Universal Robots URScript: dus_init.script

# =============================================================================
#  dus_init.script — dusan_v1
#  파라미터를 읽고 피치·행수를 계산한다. 실시간 발행 스레드를 띄운다
#
#  펜던트에서 "1_init" 자리에 스크립트 노드를 파일(File) 모드로 넣고 지정한다.
#
#  ※ def main() 으로 감싸지 말 것 (펜던트가 호출하지 않는다)
#  ※ 최상위에 global 을 쓰지 말 것 (preamble 이 이미 선언·대입해 뒀다)
#  ※ if / while 은 반드시 end 로 닫을 것
# =============================================================================

def ini_w1(a, v):
    if (v > 32000):
        v = 32000
    end
    if (v < -32000):
        v = -32000
    end
    write_port_register(a, floor(v + 0.5))
end


# 로봇 자체 레지스터 384~389 와 같은 단위.  길이 0.1mm, 회전 mRad
def ini_w6(a, p):
    ini_w1(a, p[0] * 10000)
    ini_w1(a + 1, p[1] * 10000)
    ini_w1(a + 2, p[2] * 10000)
    ini_w1(a + 3, p[3] * 1000)
    ini_w1(a + 4, p[4] * 1000)
    ini_w1(a + 5, p[5] * 1000)
end


# 절대 TCP(260~265) 는 항상 발행한다. 원점기준 상대좌표(280~285)는
# 실제 ㄹ자 스캔 중(state=4)에만 내보내고, 그 외(3점측정/원점복귀/대기/
# 완료)에는 [0,0,0,0,0,0]을 쏜다. state는 이 배경 스레드 밖에서
# write_port_register(290, ...)로만 바뀌므로 읽어서 확인한다.
#
# 위치는 베이스 좌표계 그대로 빼서 쓴다(cur - zero). 원래는
# pose_trans(zero_inv, cur_pose)로 툴 좌표계 기준값을 냈는데, 툴이
# 벽을 비스듬히 보고 있으면 베이스 Z+ 로 올라가도 이 값의 Z 성분이
# 음수로 커지는 문제가 있었다. register_map.txt 4항의 역변환 공식
# base = R_zero * rel_tcp 은 rel_tcp = R_zero^T * (cur-zero) 이므로
# 결국 cur - zero 와 정확히 같다(회전행렬을 걸었다 다시 푸는 셈).
# 그러니 처음부터 베이스 좌표계로 빼면 회전행렬 없이 같은 결과이고,
# 세로(Z)가 위로 갈수록 커지도록 직관과도 맞는다.
def pub_rel():
    global cur_pose
    global rel_pose
    global alive
    cur_pose = get_actual_tcp_pose()
    ini_w6(260, cur_pose)
    if (zero_ok == True and read_port_register(290, True) == 4):
        rel_pose = [cur_pose[0] - zero_pose[0],
                    cur_pose[1] - zero_pose[1],
                    cur_pose[2] - zero_pose[2],
                    cur_pose[3] - zero_pose[3],
                    cur_pose[4] - zero_pose[4],
                    cur_pose[5] - zero_pose[5]]
        ini_w6(280, rel_pose)
    else:
        ini_w6(280, [0, 0, 0, 0, 0, 0])
    end
    alive = alive + 1
    if (alive > 30000):
        alive = 0
    end
    write_port_register(293, alive)
end


# 제어주기마다 도는 발행 스레드. 이 뒤로는 평범한 movel 을 써도
# 이동 중 좌표가 계속 나간다.
def pub_thread():
    while (True):
        pub_rel()
        sync()
    end
end


# ------------------------------------------------------------------ 본문
# 266 = 1 이면 외부(Modbus)가 준 값을, 0 이면 펜던트 변수값을 쓴다
if (read_port_register(266, True) == 1):
    app_width = read_port_register(256, True)
    app_height = read_port_register(257, True)
    scan_h = read_port_register(258, True)
    overlap = read_port_register(259, True)
end

if (app_width <= 0):
    app_width = 1000
end
if (app_height < 0):
    app_height = 0
end
if (scan_h <= 0):
    scan_h = 200
end
if (overlap < 0):
    overlap = 0
end
if (overlap >= scan_h):
    overlap = scan_h - 10
end

# ---- 속도 : 외부(UI)가 306/307 에 쓴 값을 받는다 -----------------------
# 306 = 작업 속도 [mm/s]. movel 의 v 로 쓴다. 0 이면 변수값을 유지한다.
# 307 = 로봇 자체 속도 비율 [%] 2~100. 모든 이송 속도에 곱한다.
spd_in = read_port_register(306, True)
if (spd_in > 0):
    v_move = spd_in / 1000.0
end

spd_ratio = read_port_register(307, True)
if (spd_ratio < 2):
    spd_ratio = 100
end
if (spd_ratio > 100):
    spd_ratio = 100
end
v_move = v_move * spd_ratio / 100.0
v_scan = v_scan * spd_ratio / 100.0
v_seek = v_seek * spd_ratio / 100.0

# ---- 기준 위치 : 308 이 1 이면 310~321 의 값을 쓴다 --------------------
# 310~315 홈 관절값 [mRad], 316~321 시작 pose (길이 0.1mm, 회전 mRad)
if (read_port_register(308, True) == 1):
    Home_joint = [read_port_register(310, True) / 1000.0,
                  read_port_register(311, True) / 1000.0,
                  read_port_register(312, True) / 1000.0,
                  read_port_register(313, True) / 1000.0,
                  read_port_register(314, True) / 1000.0,
                  read_port_register(315, True) / 1000.0]
    start_pose = [read_port_register(316, True) / 10000.0,
                  read_port_register(317, True) / 10000.0,
                  read_port_register(318, True) / 10000.0,
                  read_port_register(319, True) / 1000.0,
                  read_port_register(320, True) / 1000.0,
                  read_port_register(321, True) / 1000.0]
    Home_pose = get_forward_kin(Home_joint)
end

# 상승 피치 = 스캐너 높이 - 겹침 (고정)
pitch = scan_h - overlap
if (pitch <= 0):
    pitch = 10
end

# 스캐너가 한 자리에서 scan_h 를 훑으므로
# 마지막 패스가 (높이 - scan_h) 이상이면 사각형 전체가 덮인다
rows = ceil((app_height - scan_h) * 1.0 / pitch) + 1
if (rows < 1):
    rows = 1
end
if (rows > 200):
    popup(s = "ROWS OVER LIMIT(200). CHECK HEIGHT/SCAN_H/OVERLAP", title = "dusan_v1", blocking = True)
    write_port_register(290, 9)
    halt()
end

row_idx = 0
dir_sign = 1
pass_done = 0
path_len = 0
alive = 0
zero_ok = False
n_probe = 0
n_hit = 0
qa = 0
qb = 0
qc = 0

write_port_register(290, 0)
write_port_register(291, 0)
write_port_register(292, rows)
write_port_register(293, 0)
write_port_register(294, 0)
write_port_register(295, 0)
write_port_register(296, pitch)
write_port_register(297, 0)
write_port_register(298, 0)
write_port_register(304, 0)
write_port_register(305, 0)

# 실시간 발행 스레드 기동
pub_h = start_thread(pub_thread, (), detach_mode = True)
